PROGRAM MAIN
VAR
	eStatus : E_CRANE_STATUS;
	eMode : E_Mode;
	aEndStopMessages : ARRAY[0..2] OF STRING := ['END STOP NOT ACTIVE' , 'PISTON HAS REACHED UPPER END STOP', 'PISTON HAS REACHED LOWER END STOP'];
	sEndStopMessage : STRING;
END_VAR


IF input.bEnableSwitch = FALSE THEN
output.bRunningLight := FALSE;
input.bStartSwitch := FALSE;
output.rCylinderVel := 0;
eStatus := E_Crane_Status.Unnabled;
END_IF



// Status message on HMI
IF input.bEnableSwitch = TRUE AND input.bStartSwitch = FALSE THEN
	eStatus := E_Crane_Status.Ready;
END_IF





IF input.bStartSwitch = FALSE THEN
	output.bRunningLight := FALSE;
	parameter.rRunTime := 0;
ELSIF input.bStartSwitch = TRUE THEN
	output.bRunningLight := TRUE;
	parameter.rRunTime := parameter.rRunTime + parameter.rCycleTime;
	eStatus := E_Crane_Status.Running;
END_IF





// Mode display on HMI
IF input.bModeSwitch = TRUE THEN
	eMode := E_mode.Auto;
ELSE
	eMode := E_Mode.Manual;
END_IF


// Set new max stroke
IF input.bSetNewMaxStrokeSwitch = TRUE THEN
	parameter.stStrokeRange.rCylinderStrokeMax :=Set_New_Max_Stroke(rNewMaxStroke := input.rSetInputMaxStroke);
	

input.bSetNewMaxStrokeSwitch := FALSE;
END_IF




// ENDSTOP MESSAGE
IF output.rCylinderPos >= parameter.stStrokeRange.rCylinderStrokeMax THEN
	sEndStopMessage := aEndStopMessages[1];
ELSIF output.rCylinderPos <= parameter.stStrokeRange.rCylinderStrokeMin THEN
	sEndstopMessage := aEndStopMessages[2];
ELSE
		sEndStopMessage := aEndStopMessages[0];
END_IF




// Manual Mode
IF input.bStartSwitch = TRUE AND input.bModeSwitch = FALSE THEN
	parameter.rAutoTime := 0;
	output.rCylinderPos := parameter.rRefCylinderPos;
END_IF




// AUTOMODE
IF input.bStartSwitch = TRUE
AND input.bModeSwitch = TRUE
THEN

	parameter.rInitialStrokePosition := parameter.rRefCylinderPos;
	
	// If stroke is maxed out:
	IF output.rCylinderPos >= parameter.stStrokeRange.rCylinderStrokeMax AND parameter.rRefCylinderVel > 0 THEN
		parameter.rAutoTime := 0;
		output.rCylinderVel := 0;
		
	
	// If piston is at bottom position:
	ELSIF output.rCylinderPos <= parameter.stStrokeRange.rCylinderStrokeMin AND parameter.rRefCylinderVel < 0 THEN
		parameter.rAutoTime := 0;
		output.rCylinderVel := 0;
		
	
	// When piston is between max and min:
	ELSE
		parameter.rAutoTime := parameter.rAutoTime + parameter.rCycleTime;
		output.rCylinderVel := parameter.rRefCylinderVel;
	
	END_IF
	
	output.rCylinderPos := parameter.rInitialStrokePosition + output.rCylinderVel * parameter.rAutoTime;
	parameter.rRefCylinderPos := output.rCylinderPos;
END_IF

END_PROGRAM

(* stored: Version 1.1.0.1, ProductVersion 3.1.4024.10
   POU MAIN: Id {137cafa2-2b3c-4fcc-93f3-1db729ff8b9d}, SpecialFunc None *)
